PROGRAM Lamp
VAR
	counter11 : int;
END_VAR

counter11 := counter11 + 1;

END_PROGRAM

(* stored: Version 1.1.0.1, ProductVersion 3.1.4024.12
   POU Lamp: Id {6ff10d14-b38e-48d3-97d9-6388932f2332}, SpecialFunc None *)
